{region '#Template'}
	{attribute 'Version' := '5.1.1.0'}
	{attribute 'Tags' := '"LCID": "1031", "Text": "DUT, Types, Publisher, Subscriber, RA, General, Building, Sunblind"'}
	{attribute 'Tags' := '"LCID": "1033", "Text": "DUT, Types, Publisher, Subscriber, RA, General, Building, Sunblind"'}
	{attribute 'Description' := '"LCID": "1031", "Text": "Gebäudedaten/-status für die Raumautomation - Sonnenschutz"'}
	{attribute 'Description' := '"LCID": "1033", "Text": "Building-data/-states for room-automation - Sun-protection"'}
{endregion}
TYPE ST_BA_BuildingSunblind :
STRUCT
	stSunBld						: ST_BA_SunBld;	//  Telegram for	1)	burglary, fire, ice (building-wise)
	bGlobalThAuto_Release			: BOOL;
	bGlobalTwiLgtAuto_Release		: BOOL;
	bGlobalResetManMode				: BOOL;	
   {attribute 'hide'}
	nDummy							: BYTE; 		// padding byte, in order to reach a limit corresponding to the largest data type (divisible by 8 bytes)
	nSunPrtc_PositionInterval		: UDINT;
END_STRUCT
END_TYPE

(* stored: Version 1.1.0.1, ProductVersion 3.1.4024.12
   DUT ST_BA_BuildingSunblind: Id {6ae73158-5d27-4399-8399-9948e4995717} *)
